    if (not rq_wait_for_force_reached([0, 0, 1, 0, 0, 0], [0, 0, 1, 0, 0, 0], 1, 30)):
      $ 117 "'Wait until force and torque are reached.'" "noBreak"
      # 'Wait until force and torque are reached.'
    end
    # end: URCap Program Node
    #ft mode node children finished
    kill_thread(node_execution_thread)
    #ft mode node finished
    # end: URCap Program Node
    $ 118 "MoveL"
    $ 119 "Direction: Base Y+"
    global move_thread_flag_119=0
    thread move_thread_119():
      enter_critical
      move_thread_flag_119 = 1
      local towardsPos=calculate_point_to_move_towards(p[0.0,0.0,0.0,0.0,0.0,0.0], [0.0,1.0,0.0], 0.35)
      movel(towardsPos, a=1.2, v=0.045, r=0.005)
      move_thread_flag_119 = 2
      exit_critical
    end
    move_thread_flag_119 = 0
    move_thread_han_119 = run move_thread_119()
    while (True):
      sleep(1.0E-10)
      if (move_thread_flag_119 > 1):
        join move_thread_han_119
        $ 120 "Until (distance)"
        break
      end
      sync()
    end
    $ 121 "Direction: Base X+"
    global move_thread_flag_121=0
    thread move_thread_121():
      enter_critical
      move_thread_flag_121 = 1
      local towardsPos=calculate_point_to_move_towards(p[0.0,0.0,0.0,0.0,0.0,0.0], [1.0,0.0,0.0], 0.36)
      movel(towardsPos, a=1.2, v=0.045, r=0.005)
      move_thread_flag_121 = 2
      exit_critical
    end
    move_thread_flag_121 = 0
    move_thread_han_121 = run move_thread_121()
    while (True):
      sleep(1.0E-10)
      if (move_thread_flag_121 > 1):
        join move_thread_han_121
        $ 122 "Until (distance)"
        break
      end
      sync()
    end
    $ 123 "Direction: Base Y-"
    global move_thread_flag_123=0
    thread move_thread_123():
      enter_critical
      move_thread_flag_123 = 1
      local towardsPos=calculate_point_to_move_towards(p[0.0,0.0,0.0,0.0,0.0,0.0], [0.0,-1.0,0.0], 0.35)
      movel(towardsPos, a=1.2, v=0.045, r=0.005)
      move_thread_flag_123 = 2
      exit_critical
    end
    move_thread_flag_123 = 0
    move_thread_han_123 = run move_thread_123()
    while (True):
      sleep(1.0E-10)
      if (move_thread_flag_123 > 1):
        join move_thread_han_123
        $ 124 "Until (distance)"
        break
      end
      sync()
    end
    $ 125 "Direction: Base X-"
    global move_thread_flag_125=0
    thread move_thread_125():
      enter_critical
      move_thread_flag_125 = 1
      local towardsPos=calculate_point_to_move_towards(p[0.0,0.0,0.0,0.0,0.0,0.0], [-1.0,0.0,0.0], 0.36)
      movel(towardsPos, a=1.2, v=0.045)
      move_thread_flag_125 = 2
      exit_critical
    end
    move_thread_flag_125 = 0
    move_thread_han_125 = run move_thread_125()
    while (True):
      sleep(1.0E-10)
      if (move_thread_flag_125 > 1):
        join move_thread_han_125
        $ 126 "Until (distance)"
        break
      end
      sync()
    end
    $ 127 "MoveL"
    $ 128 "Direction: Base Z+"
    global move_thread_flag_128=0
    thread move_thread_128():
      enter_critical
      move_thread_flag_128 = 1
      local towardsPos=calculate_point_to_move_towards(p[0.0,0.0,0.0,0.0,0.0,0.0], [0.0,0.0,1.0], 0.025)
      movel(towardsPos, a=1.2, v=0.06)
      move_thread_flag_128 = 2
      exit_critical
    end
    move_thread_flag_128 = 0
    move_thread_han_128 = run move_thread_128()
    while (True):
      sleep(1.0E-10)
      if (move_thread_flag_128 > 1):
        join move_thread_han_128
        $ 129 "Until (distance)"
        break
      end
      sync()
    end
    # begin: URCap Program Node
    #   Source: Robotiq_Copilot, 1.22.1.14215, Robotiq Inc.
    #   Type: Finishing Tool Control
    $ 130 "Stop tool"
    set_standard_digital_out(0, False)
    # end: URCap Program Node
  end
  thread EventThread():
    while (True):
      if (get_standard_digital_in(1) !=   True  ):
        $ 34 "Set DO[0]=Off"
        set_standard_digital_out(0, False)
        set_tcp(p[0.0,0.0,0.105,0.0,0.0,0.0])
        $ 35 "Set DO[1]=Off"
        set_standard_digital_out(1, False)
        set_tcp(p[0.0,0.0,0.105,0.0,0.0,0.0])
        $ 36 "Halt"
        halt
      end
      sync()
    end
  end
  eventThread = run EventThread()
  while (True):
    $ 2 "Robot Program"
    $ 3 "count≔count+1"
    global count=count+1
    $ 4 "Loop"
    while (True):
      $ 5 "Wait DI[0]=HI"
      while (get_standard_digital_in(0) == False):
        sync()
      end
      $ 6 "Set DO[1]=On"
      set_standard_digital_out(1, True)
      set_tcp(p[0.0,0.0,0.105,0.0,0.0,0.0])
      $ 7 "MoveJ"
      $ 8 "End" "breakAfter"
      movej(get_inverse_kin(pose_trans(Point_1, pose_trans(p[-.675004262635, .184662326493, -.049942421086, .000133991792, -.000000000005, 3.141592635831], End_p)), qnear=End_q), a=1.3962634015954636, v=1.0471975511965976)
      $ 9 "MoveJ"
      $ 10 "Ready" "breakAfter"
      set_tcp(p[0.0,0.0,0.105,0.0,0.0,0.0])
      movej(get_inverse_kin(pose_trans(Point_1, pose_trans(p[-.728914284199, .189000000000, -.030364426394, .000032022609, .000000000019, 3.141592653427], Ready_p)), qnear=Ready_q), a=1.3962634015954636, v=1.0471975511965976)
      $ 11 "Call sandTop"
      sandTop()
      $ 12 "Call positionFace1"
      positionFace1()
      $ 13 "Call sandFace"
      sandFace()
      $ 14 "MoveJ"
      $ 15 "Waypoint_3" "breakAfter"
      movej(get_inverse_kin(pose_trans(Point_1, pose_trans(p[-.728914284199, .189000000000, -.030364426394, .000032022609, .000000000019, 3.141592653427], Waypoint_3_p)), qnear=Waypoint_3_q), a=1.3962634015954636, v=1.0471975511965976)
      $ 16 "Call sandFace"
      sandFace()
      $ 17 "MoveJ"
      $ 18 "Waypoint_4" "breakAfter"
      movej(get_inverse_kin(pose_trans(Point_1, pose_trans(p[-.728914284199, .189000000000, -.030364426394, .000032022609, .000000000019, 3.141592653427], Waypoint_4_p)), qnear=Waypoint_4_q), a=1.3962634015954636, v=1.0471975511965976)
      $ 19 "Waypoint_5" "breakAfter"
      movej(get_inverse_kin(pose_trans(Point_1, pose_trans(p[-.585004860076, .315000000003, -.056950098208, .000133991792, -.000000000086, 3.141592635831], Waypoint_5_p)), qnear=Waypoint_5_q), a=1.3962634015954636, v=1.0471975511965976)
      $ 20 "Call sandFace_1"
      sandFace_1()
      # begin: URCap Program Node
      #   Source: Robotiq_Copilot, 1.22.1.14215, Robotiq Inc.
      #   Type: Finishing Tool Control
      $ 21 "Stop tool"
      set_standard_digital_out(0, False)
      # end: URCap Program Node
      $ 22 "MoveJ"
      $ 23 "Waypoint_7" "breakAfter"
      movej(get_inverse_kin(Waypoint_7_p, qnear=Waypoint_7_q), a=1.3962634015954636, v=1.0471975511965976)
      $ 24 "MoveJ"
      $ 25 "BackClear" "breakAfter"
      movej(get_inverse_kin(pose_trans(Point_1, pose_trans(p[-.585004860076, .315000000003, -.056950098208, .000133991792, -.000000000086, 3.141592635831], BackClear_p)), qnear=BackClear_q), a=1.3962634015954636, v=1.0471975511965976)
      $ 26 "Call sandBack"
      sandBack()
      $ 27 "MoveJ"
      $ 28 "End" "breakAfter"
      movej(get_inverse_kin(pose_trans(Point_1, pose_trans(p[-.675004262635, .184662326493, -.049942421086, .000133991792, -.000000000005, 3.141592635831], End_p)), qnear=End_q), a=1.3962634015954636, v=1.0471975511965976)
      $ 29 "Set DO[1]=Off"
      set_standard_digital_out(1, False)
      set_tcp(p[0.0,0.0,0.105,0.0,0.0,0.0])
    end
    $ 30 "If count≟20"
    if (count == 20):
      $ 31 "Popup: change sand paper"
      popup("change sand paper", "Message", False, False, blocking=True)
      $ 32 "count≔count+1"
      global count=count+1
    end
  end
end
